{attribute 'pack_mode' := '0'}
TYPE ACMethodDischargingR EXTENDS ACMethodBaseR :
STRUCT
	//Istmenge
	_ActualQuantity : LREAL;
	//Gesamtgewicht
	_ScaleTotalWeight : LREAL;
	//Entleerzeit
	_DischargingTime : TIME;
END_STRUCT
END_TYPE

(* stored: Version 1.1.0.1, ProductVersion 3.1.4020.12
   DUT ACMethodDischargingR: Id {6b64a04f-6d09-4aab-b633-7ff29a273416} *)
